TYPE st_MaschParameter :
STRUCT
	sName		:STRING;

	bWert		:BOOL;
	nWert		:LREAL;
	tWert		:TIME;
END_STRUCT
END_TYPE

(* stored: Version 1.1.0.1
   DUT st_MaschParameter: Id {f393c68a-71b9-4f47-922b-801bb8ebd6ba} *)
